Fanuc KAREL source: kt00379.KL

-- PROVISIONAL review KL for V1013-1; original PC SHA256 309446105c9a25be37532b320835603bfa580d22dea6d1c95f141907dc7cabbd
-- Incomplete behavior may be omitted. Consult companion uncertainty JSON. Do not deploy.
PROGRAM KT00379
%NOLOCKGROUP
VAR
  I2 : INTEGER
  OUT : BOOLEAN
-- UNRESOLVED_DECL H1 type=002017
BEGIN
  -- UNRESOLVED_PC offsets 5-19; opcodes 2E,22,9D,33,B4
  -- UNRESOLVED_PC offsets 24-35; opcodes 2E,23
  -- UNRESOLVED_PC offsets 40-62; opcodes 22,9D,33,B3,21,5A,23
  -- UNRESOLVED_PC offsets 67-71; opcodes 7F
END KT00379
